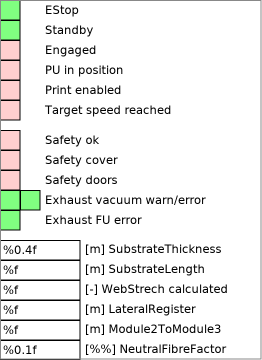
VISUALIZATION _VISU_MachineIn  // 262x360
VAR_IN_OUT
	ref : ST_ModuleMachineInterface_IN;
END_VAR
    Rectangle (0,300 80x20), "%f", text variable: ref.fLateralRegister
    Rectangle (82,300 180x18), "[m] LateralRegister"
    Rectangle (0,240 80x20), "%0.4f", text variable: ref.fSubstrateThickness
    Rectangle (82,240 180x18), "[m] SubstrateThickness"
    Rectangle (0,260 80x20), "%f", text variable: ref.fSubstrateLen
    Rectangle (82,260 180x18), "[m] SubstrateLength"
    Rectangle (0,280 80x20), "%f", text variable: ref.fWebStretchCalculated
    Rectangle (82,280 180x18), "[-] WebStrech calculated"
    Rectangle (0,320 80x20), "%f", text variable: ref.fModule2ToModule3
    Rectangle (82,320 180x18), "[m] Module2ToModule3"
    Rectangle (0,340 80x20), "%0.1f", text variable: ref.fNeutralFibreFactor
    Rectangle (82,340 180x18), "[%%] NeutralFibreFactor"
    Rectangle (42,20 180x20), "Standby"
    RoundedRectangle (0,0 20x20), colour toggle: ref.bEStop
    Rectangle (42,0 180x20), "EStop"
    RoundedRectangle (0,20 20x20), colour toggle: ref.bSleep
    RoundedRectangle (0,150 20x20), colour toggle: ref.bSafetyCoverOk
    Rectangle (42,150 180x20), "Safety cover"
    RoundedRectangle (0,170 20x20), colour toggle: ref.bServiceDoorsOk
    Rectangle (42,170 180x20), "Safety doors"
    RoundedRectangle (0,190 20x20), colour toggle: ref.bExhaustVacuumWarning
    Rectangle (42,190 180x20), "Exhaust vacuum warn/error"
    Rectangle (42,210 180x20), "Exhaust FU error"
    Rectangle (42,130 180x20), "Safety ok"
    RoundedRectangle (0,130 20x20), colour toggle: ref.bSafetyOk
    RoundedRectangle (20,190 20x20), colour toggle: ref.bExhaustVacuumError
    RoundedRectangle (0,210 20x20), colour toggle: ref.bExhaustFUError
    Rectangle (42,60 180x20), "PU in position"
    RoundedRectangle (0,60 20x20), colour toggle: ref.bUnitInPrintPosition
    Rectangle (42,40 180x20), "Engaged"
    RoundedRectangle (0,40 20x20), colour toggle: ref.bEngaged
    Rectangle (42,80 180x20), "Print enabled"
    RoundedRectangle (0,80 20x20), colour toggle: ref.bPrintEnabled
    Rectangle (42,100 180x20), "Target speed reached"
    RoundedRectangle (0,100 20x20), colour toggle: ref.bTargetSpeedReached
END_VISUALIZATION

(* stored: Version 1.1.0.1, ProductVersion 3.1.4024.11
   Visu _VISU_MachineIn: Id {0059cfba-13d6-4f84-ac2c-c60fcbba3169} *)
